{attribute 'qualified_only'}
{attribute 'strict'}
{attribute 'to_string'}
TYPE enum_states :
(
	error, // rot blinken
	stop, // Rot, Gelb blinkem
	off, // Rot leuchten
	init, // Grün blinken
	production, // grün leuchten
	ready, // gelb, grün blinken
	done, // geld, grün leuchten
	setup // gelb blinken
);
END_TYPE

(* stored: Version 1.1.0.1
   DUT enum_states: Id {e48e9dd6-550f-4d94-b517-a818feddb085} *)
